(* CoDeSys 2.3.9.31 project: CJL13.pro *)
(* Libraries: TcBase.lib 14.5.09 11:14:08, TcSystem.lib 27.2.12 14:08:36, TcUtilities.lib 10.1.13 19:12:12, TcBABasic.lib 29.10.09 13:26:44, STANDARD.LIB 5.6.98 11:03:02 *)

(* Task configuration *)
TASK Standard (PRIORITY := 0, INTERVAL := T#10ms);
	MAIN
END_TASK

(* Global variable list: Global_Variables *)
VAR_GLOBAL
	AllLightsOn: BOOL;
	AllLightsOff: BOOL;

	PushButton_Gang_A: FB_Toggle;
	PushButton_Gang_B: FB_Click;
	PushButton_Gang_C: FB_Toggle;
	PushButton_Gang_D: FB_Click;

	LED_Rolluik_Voorgevel_Up AT %Q*: BOOL;  (*Terugkoppeling status neersignaal*)
	LED_Rolluik_Voorgevel_Down AT %Q*: BOOL; (*Terugkoppeling status neersignaal*)

END_VAR

(* Global variable list: Input_variables *)
VAR_GLOBAL
	DK_Gang_A AT %I*: BOOL;
	DK_Gang_B AT %I*: BOOL;
	DK_Gang_C AT %I*: BOOL;
	DK_Gang_D AT %I*: BOOL;
	DK_Voordeur_BEL AT %I*: BOOL;

(* centrale kolom keuken *)
	DK_Kolom1_A  AT %I*: BOOL;
	DK_Kolom1_B  AT %I*: BOOL;
	DK_Kolom1_C  AT %I*: BOOL;
	DK_Kolom1_D  AT %I*: BOOL;
	DK_Kolom1_E  AT %I*: BOOL;
	DK_Kolom1_F  AT %I*: BOOL;

	DK_Kolom2_A  AT %I*: BOOL;
	DK_Kolom2_B  AT %I*: BOOL;
	DK_Kolom2_C  AT %I*: BOOL;
	DK_Kolom2_D  AT %I*: BOOL;
	DK_Kolom2_E  AT %I*: BOOL;
	DK_Kolom2_F  AT %I*: BOOL;


END_VAR

(* Global variable list: Output_variables *)
VAR_GLOBAL
	L_Eiland AT %Q*:BOOL; (*Deltalight profiel boven eiland*)
	L_Living AT %Q*:BOOL; (*Licht living*)
	L_Kelder AT %Q*:BOOL; (*Licht kelder*)
	L_Gang_GLV 	AT %Q*:BOOL;
	L_Toilet AT %Q*:BOOL;
	L_3 AT %Q*:BOOL; (* Licht bureau *)
	Rolluik_Voorgevel_Up AT %Q*: BOOL;
	Rolluik_Voorgevel_Down AT %Q*: BOOL;
	Deurbel AT %Q*:BOOL;
	L_2 AT %Q*:UINT; (*Licht boven de eettafel*)
	L_2Status AT %Q*:BOOL; (*Terugkoppeling van de status voor het licht boven de eettafel *)
	L_9 AT %Q*:UINT; (*Licht boven de eettafel*)
	L_9Status AT %Q*:BOOL; (*Terugkoppeling van de status voor het licht boven de eettafel *)
	HealthBox AT %Q*: BOOL; (* Renson Healthbox *)
END_VAR

(* Global variable list: PushButtons *)
VAR_GLOBAL

	Button_Kolom1_A : FB_Click;
(*	DK_Kolom1_B *)
	Button_Kolom1_C: FB_Click;
	Button_Kolom1_D: FB_Click;
	Button_Kolom1_E: FB_Click;
	Button_Kolom1_F: FB_Click;

	Button_Kolom2_B: FB_Click;

END_VAR

(* Global variable list: TwinCAT_Configuration *)
(* Generated automatically by TwinCAT - (read only) *)
VAR_CONFIG
	.LED_Rolluik_Voorgevel_Up AT %QX12.0 : BOOL;
	.LED_Rolluik_Voorgevel_Down AT %QX12.1 : BOOL;
	.DK_Gang_A AT %IX8.0 : BOOL;	(*  ~ {LinkedWith:TIID^Device 1 (CX1100)^CX1100-KB^Term 2 (KL1859)^Channel 1^Input} *)
	.DK_Gang_B AT %IX8.1 : BOOL;	(*  ~ {LinkedWith:TIID^Device 1 (CX1100)^CX1100-KB^Term 2 (KL1859)^Channel 2^Input} *)
	.DK_Gang_C AT %IX4.0 : BOOL;	(*  ~ {LinkedWith:TIID^Device 1 (CX1100)^CX1100-KB^Term 2 (KL1859)^Channel 3^Input} *)
	.DK_Gang_D AT %IX4.1 : BOOL;	(*  ~ {LinkedWith:TIID^Device 1 (CX1100)^CX1100-KB^Term 2 (KL1859)^Channel 4^Input} *)
	.DK_Voordeur_BEL AT %IX12.0 : BOOL;	(*  ~ {LinkedWith:TIID^Device 1 (CX1100)^CX1100-KB^Term 2 (KL1859)^Channel 6^Input} *)
	.DK_Kolom1_A AT %IX16.0 : BOOL;	(*  ~ {LinkedWith:TIID^Device 1 (CX1100)^CX1100-KB^Term 3 (KL1809)^Channel 1^Input} *)
	.DK_Kolom1_B AT %IX16.1 : BOOL;	(*  ~ {LinkedWith:TIID^Device 1 (CX1100)^CX1100-KB^Term 3 (KL1809)^Channel 2^Input} *)
	.DK_Kolom1_C AT %IX16.2 : BOOL;	(*  ~ {LinkedWith:TIID^Device 1 (CX1100)^CX1100-KB^Term 3 (KL1809)^Channel 3^Input} *)
	.DK_Kolom1_D AT %IX16.3 : BOOL;	(*  ~ {LinkedWith:TIID^Device 1 (CX1100)^CX1100-KB^Term 3 (KL1809)^Channel 4^Input} *)
	.DK_Kolom1_E AT %IX16.4 : BOOL;	(*  ~ {LinkedWith:TIID^Device 1 (CX1100)^CX1100-KB^Term 3 (KL1809)^Channel 5^Input} *)
	.DK_Kolom1_F AT %IX16.5 : BOOL;	(*  ~ {LinkedWith:TIID^Device 1 (CX1100)^CX1100-KB^Term 3 (KL1809)^Channel 6^Input} *)
	.DK_Kolom2_A AT %IX16.6 : BOOL;
	.DK_Kolom2_B AT %IX16.7 : BOOL;
	.DK_Kolom2_C AT %IX17.0 : BOOL;
	.DK_Kolom2_D AT %IX17.1 : BOOL;
	.DK_Kolom2_E AT %IX17.2 : BOOL;
	.DK_Kolom2_F AT %IX17.3 : BOOL;
	.L_Eiland AT %QX8.0 : BOOL;	(*  ~ {LinkedWith:TIID^Device 1 (CX1100)^CX1100-KB^Term 6 (KL2809)^Channel 5^L_Eiland} *)
	.L_Living AT %QX20.0 : BOOL;
	.L_Kelder AT %QX24.0 : BOOL;	(*  ~ {LinkedWith:TIID^Device 1 (CX1100)^CX1100-KB^Term 6 (KL2809)^Channel 16^Output} *)
	.L_Gang_GLV AT %QX36.0 : BOOL;	(*  ~ {LinkedWith:TIID^Device 1 (CX1100)^CX1100-KB^Term 6 (KL2809)^Channel 14^Output} *)
	.L_Toilet AT %QX36.1 : BOOL;	(*  ~ {LinkedWith:TIID^Device 1 (CX1100)^CX1100-KB^Term 6 (KL2809)^Channel 13^Output} *)
	.L_3 AT %QX44.0 : BOOL;	(*  ~ {LinkedWith:TIID^Device 1 (CX1100)^CX1100-KB^Term 6 (KL2809)^Channel 2^Output} *)
	.Rolluik_Voorgevel_Up AT %QX4.0 : BOOL;	(*  ~ {LinkedWith:TIID^Device 1 (CX1100)^CX1100-KB^Term 8 (KL2012) - Triac shutter front^Channel 1^Output} *)
	.Rolluik_Voorgevel_Down AT %QX4.1 : BOOL;	(*  ~ {LinkedWith:TIID^Device 1 (CX1100)^CX1100-KB^Term 8 (KL2012) - Triac shutter front^Channel 2^Output} *)
	.Deurbel AT %QX16.0 : BOOL;	(*  ~ {LinkedWith:TIID^Device 1 (CX1100)^CX1100-KB^Term 2 (KL1859)^Channel 4^Output} *)
	.L_2 AT %QB28 : UINT;	(*  ~ {LinkedWith:TIID^Device 1 (CX1100)^CX1100-KB^Term 13 (KL2751)^Channel 1^Data Out} *)
	.L_2Status AT %QX32.0 : BOOL;
	.L_9 AT %QB40 : UINT;	(*  ~ {LinkedWith:TIID^Device 1 (CX1100)^CX1100-KB^Term 14 (KL2751)^Channel 1^Data Out} *)
	.L_9Status AT %QX42.0 : BOOL;
	.HealthBox AT %QX48.0 : BOOL;
END_VAR

(* Global variable list: Visualisation_variables *)
VAR_GLOBAL
	Visu_Licht_Beneden: BOOL;
	Visu_Licht_Living: BOOL;
	Visu_Rolluik_Voorgevel_Up: BOOL;
	Visu_Rolluik_Voorgevel_Down: BOOL;
	Visu_Deurbel: BOOL;
	Visu_Licht_Kelder: BOOL;
	Visu_Dimmer_Eettafel: BOOL;
	Visu_Dimmer_Salon: BOOL;
	Visu_Dimmer_Salon_Status : REAL;
	Visu_Dimmer_Eettafel_Status : REAL;
	Visu_Licht_Gang: BOOL;
	Visu_Licht_Toilet: BOOL;
	Visu_AllesAan: BOOL;
	Visu_AllesUit: BOOL;
	Visu_L3: BOOL; (* Licht bureau *)
	Visu_HealthBox: BOOL; (* Ventilatie *)
END_VAR

(* POU MAIN, ST *)
PROGRAM MAIN
VAR
END_VAR
Process_Inputs;
(*Werfbediening_DeVerbouwing;*)
Rolluiken;
Control_Lights;
Deurbel_Programma;
Dimmers;
Control_Lights_ST;
Ventilation;
END_PROGRAM

(* POU Process_Inputs, ST *)
PROGRAM Process_Inputs
VAR
	R_Trig_AllesUit: R_TRIG;
END_VAR
PushButton_Gang_B(ingang:= DK_Gang_B); (* linkt de fysieke input aan de functie block FB_Click *)
PushButton_Gang_D(ingang:= DK_Gang_D);
Button_Kolom1_A(ingang:= DK_Kolom1_A);
Button_Kolom1_C(ingang:= DK_Kolom1_C);
Button_Kolom1_D(ingang:= DK_Kolom1_D);
Button_Kolom1_E(ingang:= DK_Kolom1_E);
Button_Kolom1_F(ingang:= DK_Kolom1_F);

AllLightsOff := Visu_AllesUit OR PushButton_Gang_D.EenClick;
AllLightsOn := Visu_AllesAan OR PushButton_Gang_D.TweeClick;
END_PROGRAM

(* POU Rolluiken, ST *)
PROGRAM Rolluiken
VAR
	Rolluik_Voorgevel: Rolluik;

END_VAR
Rolluik_Voorgevel
(
	DrukknopOp:=  Button_Kolom1_D.EenClick,
	DrukknopNeer:= Button_Kolom1_C.EenClick,
	Tijd:= t#20s,
	UitgOp=> Rolluik_Voorgevel_Up,
	UitgNeer=>Rolluik_Voorgevel_Down );
END_PROGRAM

(* POU TestCode/Rolluik, ST *)
FUNCTION_BLOCK Rolluik
VAR_INPUT
	DrukknopOp: BOOL;
	DrukknopNeer: BOOL;
	Tijd: TIME := t#20s;
END_VAR
VAR_OUTPUT
	UitgOp: BOOL;
	UitgNeer: BOOL;
END_VAR
VAR
	Stap: INT;
	TimerOp: TON;
	TimerNeer: TON;
	rDrukknopOp: R_TRIG;
	rDrukknopNeer: R_TRIG;
END_VAR
TimerOp(IN:= Stap = 10 , PT:= Tijd , Q=> , ET=> );
TimerNeer(IN:= Stap = 20 , PT:= Tijd , Q=> , ET=> );

rDrukknopOp(CLK:= DrukknopOp , Q=> );
rDrukknopNeer(CLK:= DrukknopNeer , Q=> );

CASE Stap OF

0:
	IF rDrukknopOp.Q THEN
		Stap := 10;
	END_IF

	IF rDrukknopNeer.Q THEN
		Stap := 20;
	END_IF

10:
	IF DrukknopNeer OR TimerOp.Q  THEN
		Stap := 0;
	END_IF

20:

	IF DrukknopOp OR TimerNeer.Q THEN
		Stap := 0;
	END_IF

END_CASE


UitgOp := Stap = 10;
UitgNeer := Stap = 20;
END_FUNCTION_BLOCK

(* POU Control_Lights, FBD *)
PROGRAM Control_Lights
VAR
	FB_Licht_Kelder: FB_LightControl_Local;
	FB_Eiland: FB_LightControl_Local;
END_VAR
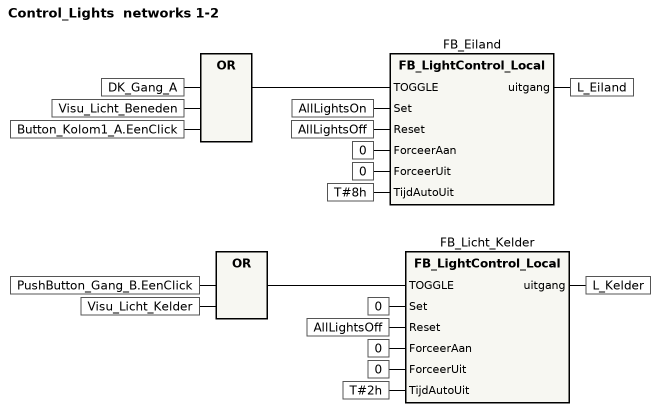
_FBD_ (* Function Block Diagram *)
NETWORK 1
	FB_Eiland:FB_LightControl_Local(TOGGLE: OR(DK_Gang_A, Visu_Licht_Beneden, Button_Kolom1_A.EenClick), Set: AllLightsOn, Reset: AllLightsOff, ForceerAan: 0, ForceerUit: 0, TijdAutoUit: T#8h) => L_Eiland
NETWORK 2
	FB_Licht_Kelder:FB_LightControl_Local(TOGGLE: OR(PushButton_Gang_B.EenClick, Visu_Licht_Kelder), Set: 0, Reset: AllLightsOff, ForceerAan: 0, ForceerUit: 0, TijdAutoUit: T#2h) => L_Kelder
_END_FBD_
(* the same logic as Structured Text *)
(* Network 1 *)
FB_Eiland(TOGGLE := DK_Gang_A OR Visu_Licht_Beneden OR Button_Kolom1_A.EenClick, Set := AllLightsOn, Reset := AllLightsOff, ForceerAan := 0, ForceerUit := 0, TijdAutoUit := T#8h);
L_Eiland := FB_Eiland.uitgang;
(* Network 2 *)
FB_Licht_Kelder(TOGGLE := PushButton_Gang_B.EenClick OR Visu_Licht_Kelder, Set := 0, Reset := AllLightsOff, ForceerAan := 0, ForceerUit := 0, TijdAutoUit := T#2h);
L_Kelder := FB_Licht_Kelder.uitgang;
END_PROGRAM

(* POU Function Blocks/FB_LightControl_Local, ST *)
FUNCTION_BLOCK FB_LightControl_Local
VAR_INPUT
	TOGGLE: BOOL;
	Set: BOOL;
	Reset: BOOL;
	ForceerAan: BOOL;
	ForceerUit: BOOL;
	TijdAutoUit: TIME;
END_VAR
VAR_OUTPUT
	uitgang: BOOL;
END_VAR
VAR
	Licht: BOOL;
	RisingEdgeToggle: R_TRIG;
	Timer1: TON;
	RisingEdgeReset: R_TRIG;
	RisingEdgeSet: R_TRIG;
END_VAR
(*====TOGGLE AAN/UIT ==================================*)
(*Toggle licht aan / uit*)
RisingEdgeToggle(CLK := Toggle );
IF (RisingEdgeToggle.Q) THEN
	Licht := NOT Licht;
END_IF


(*====AUTOMATISCH UIT OP TIJD==========================*)
Timer1(IN:= Licht AND TijdAutoUit <> T#0s, PT:= TijdAutoUit );
IF Timer1.Q THEN
	licht := FALSE;
END_IF

(*====SET/RESET===================================*)
RisingEdgeSet(CLK := Set );
IF (RisingEdgeSet.Q) THEN
	Licht := TRUE;
END_IF
RisingEdgeReset(CLK := Reset );
IF (RisingEdgeReset.Q) THEN
	Licht := FALSE;
END_IF

(*====Forceer aan/uit======================================*)
uitgang := NOT(ForceerUit) AND (ForceerAan OR Licht);
END_FUNCTION_BLOCK

(* POU Deurbel_Programma, LD *)
PROGRAM Deurbel_Programma
VAR
	Timer_Deurbel: TOF;
	Status_Deurbel: BOOL;
END_VAR
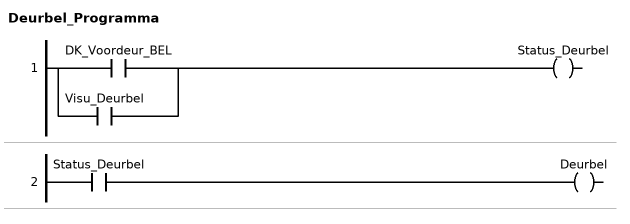
_LD_ (* Ladder Diagram *)
NETWORK 1
	{ [DK_Voordeur_BEL] | [Visu_Deurbel] } --- (Status_Deurbel)
NETWORK 2
	[Status_Deurbel] --- (Deurbel)
_END_LD_
(* the same logic as Structured Text *)
(* Network 1 *)
Status_Deurbel := DK_Voordeur_BEL OR Visu_Deurbel;
(* Network 2 *)
Deurbel := Status_Deurbel;
END_PROGRAM

(* POU Dimmers, ST *)
PROGRAM Dimmers
VAR
	Dimmer_Eettafel: FB_Dimmer1SwitchEco;
	(*Dimmer_Eettafel2: FB_Dimmer1Switch;*)
	Dimmer_SalonL9: FB_Dimmer1SwitchEco;
END_VAR
Dimmer_Eettafel
(
bSwitchDimm:= Visu_Dimmer_Eettafel OR PushButton_Gang_B.TweeClick OR DK_Kolom1_B,
tDimmTime:= t#3s,
bOn:= AllLightsOn,
bOff:= AllLightsOff,
nOut=>L_2,
bLight => L_2Status,
);

Visu_Dimmer_Salon_Status := OnAScaleOfZeroToTen(L_9);
Visu_Dimmer_Eettafel_Status := OnAScaleOfZeroToTen(L_2);

Dimmer_SalonL9
(
	bSwitchDimm:= DK_Kolom2_A OR Visu_Dimmer_Salon,
	bOn:= AllLightsOn,
	bOff:= AllLightsOff,
	tSwitchOverTime:= ,
	tDimmTime:= t#3s ,
	nOut=>L_9 ,
	bLight=>L_9Status );
END_PROGRAM

(* POU Functions/OnAScaleOfZeroToTen, ST *)
FUNCTION OnAScaleOfZeroToTen : LREAL
VAR_INPUT
	ValueIn : INT;

END_VAR
VAR
END_VAR
OnAScaleOfZeroToTen := ValueIn /  3267.6;
END_FUNCTION

(* POU Control_Lights_ST, ST *)
PROGRAM Control_Lights_ST
VAR
	FB_Light_Hallway_Downstairs: FB_Light;
	FB_Light_Toilet: FB_Light;
	FB_Light_3: FB_Light;
END_VAR
FB_Light_Hallway_Downstairs(
	bOn:= AllLightsOn ,
	bOff:=AllLightsOff ,
	bToggle:=Button_Kolom1_F.EenClick OR Visu_Licht_Gang OR DK_Gang_C
	 , bLight=> L_Gang_GLV);

FB_Light_Toilet(
	bOn:= 0 ,
	bOff:=AllLightsOff ,
	bToggle:=Button_Kolom1_E.EenClick OR Visu_Licht_Toilet
	 , bLight=> L_Toilet);


FB_Light_3(
	bOn:= AllLightsOn ,
	bOff:=AllLightsOff ,
	bToggle:=Button_Kolom1_A.TweeClick OR Visu_L3
	 , bLight=> L_3);
END_PROGRAM

(* POU Ventilation, ST *)
PROGRAM Ventilation
VAR
	FB_Ventilation_OnOff: FB_Light;
END_VAR
FB_Ventilation_OnOff(
	bOn:= 0 ,
	bOff:=0 ,
	bToggle:= Visu_HealthBox
	 , bLight=> HealthBox);
END_PROGRAM

(* POU Function Blocks/FB_Click, ST *)
FUNCTION_BLOCK FB_Click
VAR_INPUT
	Ingang				: BOOL;
END_VAR
VAR_OUTPUT
	NoChange			:BOOL;
	EenClick				: BOOL;
	TweeClick			: BOOL;
	DrieClick				: BOOL;
	LangClick			: BOOL;
END_VAR
VAR
	RisingEdgeIngang	: R_TRIG;
	FalingEdgeTimer1	: F_TRIG;
	Timer1				: TOF;
	teller				: UINT;
END_VAR
NoChange := Ingang;
IF ingang = FALSE THEN
	EenClick:= FALSE;
	TweeClick:= FALSE;
	DrieClick:= FALSE;
	LangClick:= FALSE;
END_IF;

RisingEdgeIngang(CLK:=Ingang);
Timer1(IN:= RisingEdgeIngang.Q, PT:= T#400ms);
FalingEdgeTimer1(CLK:=Timer1.Q );

IF RisingEdgeIngang.Q THEN
	teller := teller +1;
END_IF

IF FalingEdgeTimer1.Q THEN
	IF ingang THEN
		LangClick := TRUE;
	ELSE
		CASE teller OF
			1: EenClick:= TRUE;
			2: TweeClick:= TRUE;
			3: DrieClick:= TRUE;
		END_CASE
	END_IF
	teller := 0;
END_IF
END_FUNCTION_BLOCK

(* POU Function Blocks/FB_Toggle, LD *)
FUNCTION_BLOCK FB_Toggle
VAR_INPUT
	iToggle: BOOL;
END_VAR
VAR_OUTPUT
	oUitgang : BOOL;
END_VAR
VAR
	status: BOOL;
	RisingEdge: R_TRIG;
END_VAR
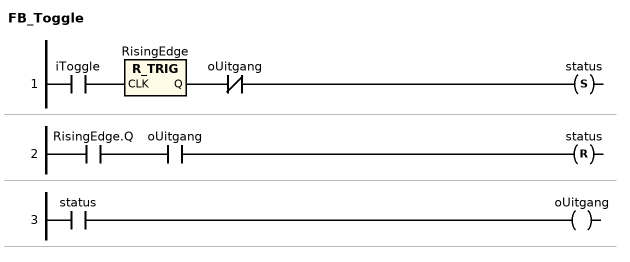
_LD_ (* Ladder Diagram *)
NETWORK 1
	[iToggle] - RisingEdge:R_TRIG(CLK: *) - [/oUitgang] --- (S status)
NETWORK 2
	[RisingEdge.Q] - [oUitgang] --- (R status)
NETWORK 3
	[status] --- (oUitgang)
_END_LD_
(* the same logic as Structured Text *)
(* Network 1 *)
RisingEdge(CLK := iToggle);
IF RisingEdge.Q AND NOT oUitgang THEN status := TRUE; END_IF;
(* Network 2 *)
IF RisingEdge.Q AND oUitgang THEN status := FALSE; END_IF;
(* Network 3 *)
oUitgang := status;
END_FUNCTION_BLOCK

(* Visualisation BENEDEN
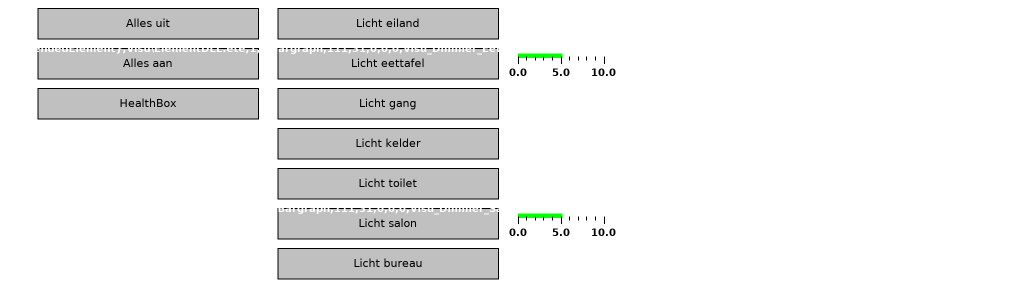
rounded rectangle at (260,70)-(481,101): text "Licht eettafel"; alarm colour if .L_2Status; taps .Visu_Dimmer_Eettafel
rounded rectangle at (260,110)-(481,141): text "Licht gang"; alarm colour if .L_Gang_GLV; taps .Visu_Licht_Gang
rounded rectangle at (260,30)-(481,61): text "Licht eiland"; alarm colour if .L_Eiland; taps .Visu_Licht_Beneden
rounded rectangle at (260,190)-(481,221): text "Licht toilet"; alarm colour if .L_Toilet; taps .Visu_Licht_Toilet
rounded rectangle at (260,150)-(481,181): text "Licht kelder"; alarm colour if .L_Kelder; taps .Visu_Licht_Kelder
rounded rectangle at (20,30)-(241,61): text "Alles uit"; alarm colour if .AllLightsOff; taps .Visu_AllesUit
rounded rectangle at (260,230)-(481,261): text "Licht salon"; alarm colour if .L_9Status; taps .Visu_Dimmer_Salon
rounded rectangle at (20,70)-(241,101): text "Alles aan"; alarm colour if .AllLightsOn; taps .Visu_AllesAan
group at (490,230)-(601,261)
  rectangle at (5,0)-(6,1): text "{ExtendedElement},Visu\ElementDLL.ete,1,@Bargraph,111,31,0,0,0,Visu_Dimmer_Salon_Status,,%.1f,1,5,0,10,0,0,0,0,0,0,0,-13,16,700,Arial,0,255,0,255,0,0,0,0,0,0,0,0,0,,0,"
  rectangle at (12,5)-(61,9): alarm colour if (Visu_Dimmer_Salon_Status) < 0; right ((Visu_Dimmer_Salon_Status * 1.0) - 5)  * 9.6
  rectangle at (0,16)-(24,28): text "0.0"
  rectangle at (48,16)-(72,28): text "5.0"
  rectangle at (91,16)-(124,28): text "10.0"
group at (490,70)-(601,101)
  rectangle at (5,0)-(6,1): text "{ExtendedElement},Visu\ElementDLL.ete,1,@Bargraph,111,31,0,0,0,Visu_Dimmer_Eettafel_Status,,%.1f,1,5,0,10,0,0,0,0,0,0,0,-13,16,700,Arial,0,255,0,255,0,0,0,0,0,0,0,0,0,,0,"
  rectangle at (12,5)-(61,9): alarm colour if (Visu_Dimmer_Eettafel_Status) < 0; right ((Visu_Dimmer_Eettafel_Status * 1.0) - 5)  * 9.6
  rectangle at (0,16)-(24,28): text "0.0"
  rectangle at (48,16)-(72,28): text "5.0"
  rectangle at (91,16)-(124,28): text "10.0"
rounded rectangle at (260,270)-(481,301): text "Licht bureau"; alarm colour if .L_3; taps .Visu_L3
rounded rectangle at (20,110)-(241,141): text "HealthBox"; alarm colour if .HealthBox; taps .Visu_HealthBox
22 more shapes without text or variables
*)
